(* PLC project Unnamed, Unknown Unnamed 1 *)
(* stored: creationDateTime 2026-02-02T15:43:33, modificationDateTime 2026-02-02T16:04:50 *)

PROGRAM program0
  VAR
    TLB1 : BOOL;
    TLB2 : BOOL;
    MV1 : BOOL;
    MV2 : BOOL;
    Start : BOOL;
    Stop : BOOL;
    CycleOn : BOOL;
    Buzzer : BOOL;
    RS0 : RS;
    SR0 : SR;
  END_VAR
  VAR  (* added by the conversion: wires and edge detectors of the diagram *)
    R_TRIG1 : R_TRIG;
    F_TRIG2 : F_TRIG;
  END_VAR

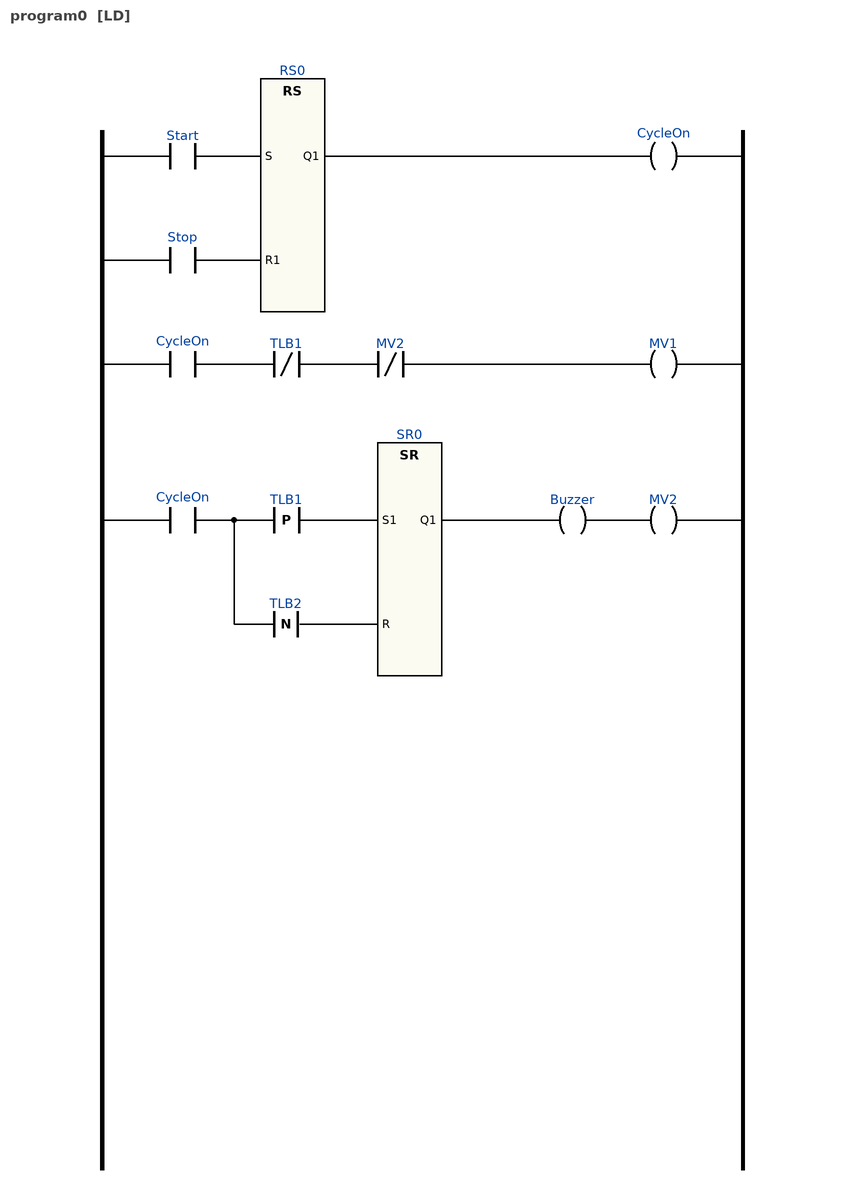
(* LD diagram, written out as Structured Text *)
RS0(S := Start, R1 := Stop);
CycleOn := RS0.Q1;
MV1 := CycleOn AND NOT TLB1 AND NOT MV2;
R_TRIG1(CLK := TLB1);
F_TRIG2(CLK := TLB2);
SR0(S1 := CycleOn AND R_TRIG1.Q, R := CycleOn AND F_TRIG2.Q);
MV2 := SR0.Q1;
Buzzer := SR0.Q1;
END_PROGRAM

CONFIGURATION Config0
  RESOURCE Res0 ON PLC
    TASK task0(INTERVAL := T#20ms, PRIORITY := 0);
    PROGRAM instance0 WITH task0 : program0;
  END_RESOURCE
END_CONFIGURATION
